{attribute 'GeneratedUsingTerminal: EK1122-0000-0018'}
{attribute addProperty BoxType "EK1122-0000-0018"}
{attribute addProperty Id "Beckhoff_EL34xxsub_EK1100EK1100_1FC0878B2"}
{attribute addProperty CRC "3216860380"}
{attribute addProperty Size "2"}
TYPE Beckhoff_EL34xxEK1122_BFBD64DC EXTENDS EK1122_1FC0878B :
STRUCT
	{attribute addProperty Name "Beckhoff_EL34xxsub_EK1100"}
	{attribute addProperty PreviousPort "Beckhoff EL34xxEK1122 : D"}
	Beckhoff_EL34xxsub_EK1100 : EK1100_1FC0878B;
END_STRUCT
END_TYPE

(* stored: Version 1.2.0.0, ProductVersion 3.1.4024.9
   DUT Beckhoff_EL34xxEK1122_BFBD64DC: Id {c5ebe975-8cea-4d04-8708-91149d0bd02c} *)
